FUNCTION_BLOCK FB_CamDTDriver	
VAR_INPUT
	Reset                                        :BOOL; //复位     
   	bCamInExecute			                :BOOL;	//凸轮耦合启动
   	bCreatTable		                        :BOOL;	//凸轮阶建启动
	iTable		                              :UINT;   //凸轮表号    
    fMainPos                                  :REAL;//叠台到位主轴的角度
    fbStartingPoint                           :REAL;//叠台凸轮的起点
	fbEndPoint								  :REAL;//叠台凸轮的终点
	fbCenterPoint								:REAL;//叠台压刀外边到过辊的中心距离
	
END_VAR
VAR_IN_OUT
	axisSlave		                    :axis_ref;  //从轴
	axisMaster		                    :axis_ref;  //主轴
	arrTableData: ARRAY[0..3600,0..1] OF LREAL;//叠台凸轮数据
END_VAR

VAR_OUTPUT
	Master_MidPos: LREAL;// 叠台压好到过辊中分主轴相位
	iFend: INT;// 叠台压刀到过辊中心主轴相位对应的索引	
    bCreatTableDone         :BOOL;//凸轮创建完成
    bCreatTableError         :BOOL;//凸轮创建错误
	bError                         :BOOL;//报警
	bReady                        :BOOL;//准备OK
	bInSync		                   :BOOL;//凸轮耦合中
END_VAR


VAR
	fbCamInSlave: MC_CamIn;
	fbCamOut: MC_CamOut;
	fbHaltSlave: MC_Halt; 
	rtrigs		:ARRAY[1..3]OF R_TRIG;
	ftrigs		:ARRAY[1..3]OF F_TRIG;
	iCamInStep: UINT;
	 PositionData			:	ARRAY[1..4] OF MC_MotionFunctionPoint;	
     PositionData1			:	ARRAY[1..4] OF MC_MotionFunctionPoint;	

	fbCamtableselect:			MC_CamTableSelect;
	Cam_table:				MC_CAM_REF;
    CamTable_MF:             MC_CAM_REF;

	rtError:  Tc2_Standard.R_TRIG;  	

    fbChangeCamModeSetOut	:	Tc2_MC2.ST_McOutputs;

	MA1: BOOL;
   fbCamInOut:                       Tc2_MC2.ST_McOutputs;
   bPoints :ARRAY[1..5] OF MC_MotionFunctionPoint; 
   mcReadMotionFunction: MC_ReadMotionFunction;
   mcReadMotionFunctionOut:Tc2_MC2.ST_McOutputs;
	iCreatTableStep: INT;
	fbHaltMaster: INT;
	bWriteCamData: BOOL;
	fSlavePos1: REAL;
	fSlavePos2: REAL;
	// 叠台移动的距离
	fBeltSpacePos: REAL;
	// 叠台中心点，主轴相位计算
	ReadPointVelues: BOOL;
	i: INT;
	Test_int: INT;
	mcReadMotionFunctionValues: MC_ReadMotionFunctionValues;
	CamTable: MC_CAM_REF;
	// 叠台凸轮数据读取完成
	arrReadPosDone: BOOL;
	rtRead: R_TRIG;
	ftRead: F_TRIG;	
	CamTable1: MC_CAM_REF;
	CamTable2: MC_CAM_REF;
	mcReadMotionFunctionValues_Busy: BOOL;
	mcReadMotionFunctionValues_Error: BOOL;
	mcReadMotionFunctionValues_ErrorID: UDINT;
	FB_ReadCamarrPos1: FB_ReadCamarrPos;
	arrReadPosDone1: BOOL;
	arrTableData1: ARRAY [0..3600, 0..1] OF LREAL;
	mcReadMotionFunctionValues1: MC_ReadMotionFunctionValues;
	CamTable3: MC_CAM_REF;
	TEST: BOOL;
END_VAR

rtrigs[1](CLK:=bCreatTable);  
ftrigs[1](CLK:=bCreatTable);  




CASE iCreatTableStep OF   
0:  
    IF  NOT bInSync  AND  rtrigs[1].Q  AND NOT bCreatTableError  THEN
         fbCamtableselect.Execute:=FALSE;
         bCreatTableDone:=FALSE;
         bCreatTable:=FALSE;
         bWriteCamData:=TRUE;
		 ReadPointVelues:=FALSE;
         iCreatTableStep:=10;
    END_IF 
10: //节点写入完成
   IF NOT bWriteCamData THEN 
	  fbCamtableselect.Execute:=TRUE;     
	 iCreatTableStep:=20;	
  END_IF
20:	//凸轮生成	
	IF NOT  fbCamtableselect.Execute     THEN
        //bCreatTableDone:=TRUE;
		iCreatTableStep:=30;	
    ELSIF  fbCamtableselect.Error THEN
       bCreatTableError:=TRUE;
       iCreatTableStep:=999;	//创建凸轮失败
	END_IF	
30:
		ReadPointVelues:=TRUE;
		IF arrReadPosDone THEN
			bCreatTableDone:=TRUE;
			ReadPointVelues:=FALSE;
			iCreatTableStep:=0;
		ELSIF mcReadMotionFunctionValues1.Error THEN
       		bCreatTableError:=TRUE;
       		iCreatTableStep:=999;	//创建凸轮失败			
		END_IF	
END_CASE	
(**********故障***********)
	IF  Reset  AND bCreatTableError  THEN  
	   bCreatTableError:=FALSE;
	   iCreatTableStep:=0;
	END_IF
(*****************************************耦合***************************************)
fbCamInSlave.BufferMode;
fbCamInSlave.Options.ActivationMode;
fbCamInSlave.Options.ActivationPosition;
fbCamInSlave.Options.ActivationMode;
fbCamInSlave.Options.InterpolationType;
fbCamInSlave.Options.MasterScalingMode;
fbCamInSlave.Options.SlaveScalingMode;

(************************************  相关状态  *************************************************)
bReady:= axisSlave.Status.ControlLoopClosed  AND axisMaster.Status.ControlLoopClosed AND  
               NOT bInSync  AND NOT bError   AND  bCreatTableDone   ;  

rtrigs[2](CLK:=bCamInExecute);  
ftrigs[2](CLK:=bCamInExecute);  

CASE iCamInStep OF
0:  
      fbCamInSlave.MasterOffset:=0;
      fbCamInSlave.SlaveOffset:=0;
      fbCamtableselect.Execute:=FALSE;
   	  fbCamInSlave.Execute:=FALSE;
	  fbCamOut.Execute:=FALSE;
	  fbHaltSlave.Execute:=FALSE;
      iCreatTableStep:=0;
      iCamInStep:=10;
10:
  IF bCamInExecute  AND  bReady THEN //耦合
	   iCamInStep:=100;
  ELSIF ftrigs[2].Q THEN  //解耦
	    iCamInStep:=200;
 ELSIF bInSync AND NOT bCamInExecute THEN
        iCamInStep:=200;
  END_IF

100:(**凸轮耦合**)
      fbCamInSlave.Execute:=TRUE;
      iCamInStep:=110;
110:
    IF NOT  fbCamInSlave.Execute AND axisSlave.Status.Coupled THEN
        bInSync:=TRUE;  //同步状态输出
        iCamInStep:=0;
   ELSIF fbCamInSlave.Error OR fbCamInSlave.CommandAborted THEN
         iCamInStep:=999;
    END_IF

(**********************解耦  *******************************)
200:
		fbCamOut.Execute:=TRUE;
		iCamInStep:=210;
210: 
	IF  NOT axisSlave.Status.Coupled   THEN 
	  	fbHaltSlave.Execute:=TRUE; 
	 	iCamInStep:=220;
    ELSIF  fbCamOut.Error  THEN
        iCamInStep:=999;
	END_IF
220: 
	IF axisSlave.Status.NotMoving    THEN
		bInSync:=FALSE; //同步状态输
		iCamInStep:=0;
     ELSIF fbHaltSlave.Error OR fbHaltSlave.CommandAborted THEN
          iCamInStep:=999;
	END_IF
END_CASE

(**********故障复位***********)
	IF  Reset  AND bError  THEN  
	   bError:=FALSE;
	   iCamInStep:=0;
	END_IF
rtError(CLK:=fbCamInSlave.Error  OR fbCamOut.Error OR fbHaltSlave.Error OR iCamInStep=999     , Q=> );
IF 	rtError.Q THEN
	bError:=TRUE;
	bInSync:=FALSE; //同步状态输
END_IF


Motion();      
ModifyCam();

ACTION ModifyCam:
//凸轮创建
fbCamtableselect(   
	Execute:=                        fbCamtableselect.Execute ,
	Periodic:=                       TRUE ,
	MasterAbsolute:=             FALSE,//
	SlaveAbsolute:=                FALSE ,//
	CamTableID:=                  iTable,
	Master:=                         axisMaster ,
	Slave:=                            axisSlave ,
	CamTable:=                     Cam_table , );
IF fbCamtableselect.Done THEN
    fbCamtableselect.Execute:=FALSE;
END_IF
//凸轮关键点写入
IF bWriteCamData  THEN    //98     初始点   90
	  Cam_table.ArraySize:=SIZEOF(PositionData1); 
	  Cam_table.NoOfColumns:=1;
	  Cam_table.NoOfRows:=3;
	  Cam_table.pArray:=ADR(PositionData1);
	  Cam_table.TableType:=MC_TABLETYPE_MOTIONFUNCTION;
  
	  fBeltSpacePos:=fbEndPoint-fbStartingPoint;
	  
	  PositionData1[1].	PointIndex	:=	        1;
	  PositionData1[1].	FunctionType	:=		MOTIONFUNCTYPE_POLYNOM7_MM;
	  PositionData1[1].	PointType	:=	        MOTIONPOINTTYPE_MOTION;
	  PositionData1[1].	RelIndexNextPoint	:=  1;
	  PositionData1[1].	MasterPos	:=	        0;
	  PositionData1[1].	SlavePos	:=	        0;		
	  PositionData1[1].	SlaveVelo	:=	        0;
	  
	  PositionData1[2].	PointIndex	:=	        2;
	  PositionData1[2].	FunctionType	:=		MOTIONFUNCTYPE_POLYNOM1;
	  PositionData1[2].	PointType	:=	        MOTIONPOINTTYPE_MOTION;
	  PositionData1[2].	RelIndexNextPoint	:=  1;
	  PositionData1[2].	MasterPos	:=	        fMainPos;
	  PositionData1[2].	SlavePos	:=	        fBeltSpacePos;	
	  PositionData1[2].	SlaveVelo	:=	        0	;
	  
	  PositionData1[3].	PointIndex	:=	        3;
	  PositionData1[3].	FunctionType	:=		MOTIONFUNCTYPE_POLYNOM7_MM;
	  PositionData1[3].	PointType	:=	        MOTIONPOINTTYPE_MOTION;
	  PositionData1[3].	RelIndexNextPoint	:=  0;
	  PositionData1[3].	MasterPos	:=	        360;
	  PositionData1[3].	SlavePos	:=	        fBeltSpacePos;	
	  PositionData1[3].	SlaveVelo	:=	       0;
   
     bWriteCamData:=FALSE;
END_IF


//读取叠台的数据
rtRead(CLK:=ReadPointVelues , Q=> );
ftRead(CLK:=ReadPointVelues , Q=> );	
	IF rtRead.Q THEN
		mcReadMotionFunctionValues.Execute:=TRUE;
		CamTable3.pArray:=ADR(arrTableData);
		CamTable3.ArraySize:=SIZEOF(arrTableData);
		CamTable3.NoOfColumns:=2;
		CamTable3.NoOfRows:=3601;
		CamTable3.TableType:=10;	
	END_IF	
	 mcReadMotionFunctionValues1(
		  Execute:=                          mcReadMotionFunctionValues.Execute , 
		  CamTableID:=                   iTable , 
		  ValueSelectMask:=               1 ,
		  StartPosMaster:=               0 , 
		  EndPosMaster:=                360 , //360
		  Increment:=                       0.1 , 
		  Done=>                           arrReadPosDone , 
		  Busy=>mcReadMotionFunctionValues_Busy                              , 
		  Error=>mcReadMotionFunctionValues_Error                             , 
		  ErrorID=>mcReadMotionFunctionValues_ErrorID                         , 
		  CamTable:=                      CamTable3      );
	IF ftRead.Q THEN
		mcReadMotionFunctionValues.Execute:=FALSE;	
	END_IF	
//叠台中心点，主轴相位计算 fbCenterPoint
	Test_int:=REAL_TO_INT(fMainPos*10);
	FOR	i:=0 TO Test_int BY 1  DO
		IF (fbCenterPoint-0.15)< arrTableData[i,1] AND arrTableData[i,1]<(fbCenterPoint +0.15) THEN
			iFend:=i;
			Master_MidPos:=arrTableData[i,0];			
		END_IF		
	END_FOR
END_ACTION

ACTION Motion:
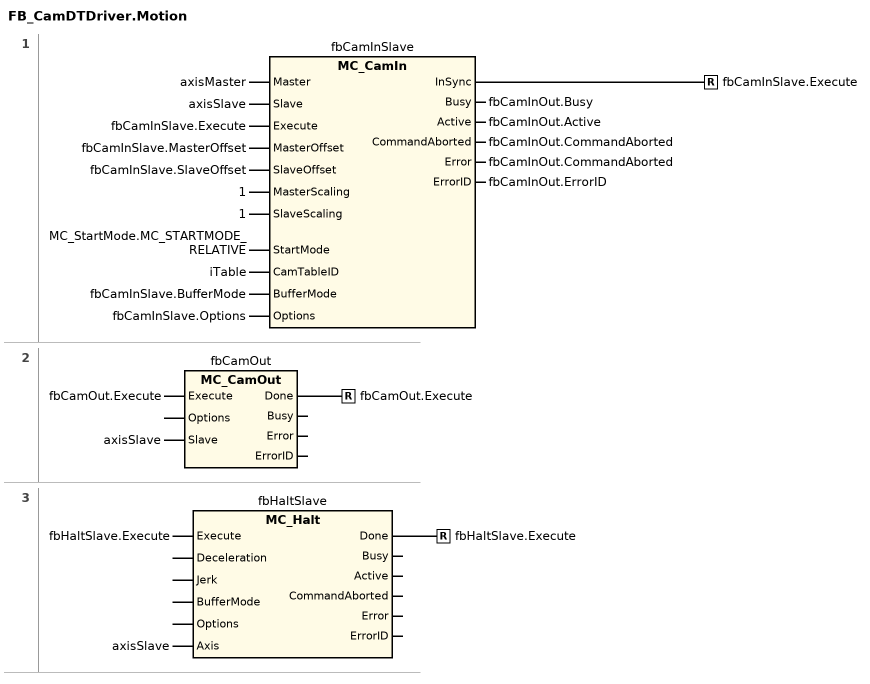
// NETWORK 1
fbCamInSlave(
    Master := axisMaster,
    Slave := axisSlave,
    Execute := fbCamInSlave.Execute,
    MasterOffset := fbCamInSlave.MasterOffset,
    SlaveOffset := fbCamInSlave.SlaveOffset,
    MasterScaling := 1,
    SlaveScaling := 1,
    StartMode := MC_StartMode.MC_STARTMODE_RELATIVE,
    CamTableID := iTable,
    BufferMode := fbCamInSlave.BufferMode,
    Options := fbCamInSlave.Options,
    Busy => fbCamInOut.Busy,
    Active => fbCamInOut.Active,
    CommandAborted => fbCamInOut.CommandAborted,
    Error => fbCamInOut.CommandAborted,
    ErrorID => fbCamInOut.ErrorID); // MC_CamIn
fbCamInSlave.Execute R= fbCamInSlave.InSync;

// NETWORK 2
fbCamOut(Execute := fbCamOut.Execute, Slave := axisSlave); // MC_CamOut
fbCamOut.Execute R= fbCamOut.Done;

// NETWORK 3
fbHaltSlave(Execute := fbHaltSlave.Execute, Axis := axisSlave); // MC_Halt
fbHaltSlave.Execute R= fbHaltSlave.Done;
END_ACTION

END_FUNCTION_BLOCK

(* stored: Version 1.1.0.1, ProductVersion 3.1.4024.9
   POU FB_CamDTDriver: Id {691e79d7-fe42-48ae-bc38-5225fb2a0e85}, SpecialFunc None
   Action ModifyCam: Id {a41f5caa-fb74-4326-8cff-abe2d4f7a6dd}
   Action Motion: Id {167d9c9a-345a-4515-a834-d57fd96a99a3} *)
